FUNCTION_BLOCK FB_GroupElement_HMI EXTENDS FB_BaseGroupElement_HMI IMPLEMENTS ITF_GroupElement_HMI
VAR
	itfGroupElementConnector			: ITF_GroupElement_HMI_Connector;
	refstGroupElementData				: REFERENCE TO ST_GroupElement_HMI;
	
	itfControlElement1					: ITF_ControlElement_HMI;
	itfControlElement2					: ITF_ControlElement_HMI;
	itfComponent1						: ITF_Component_HMI;
	itfComponent2						: ITF_Component_HMI;
	
END_VAR

METHOD FB_init : BOOL
VAR_INPUT
	bInitRetains : BOOL; // if TRUE, the retain variables are initialized (warm start / cold start)
	bInCopyCode : BOOL;  // if TRUE, the instance afterwards gets moved into the copy code (online change)
	itfBaseLoggerConnector				: ITF_BaseLogger_HMI_Connector;	//bezpośredni łącznik do logera
	itfGroupElementConnector			: ITF_GroupElement_HMI_Init;
	itfControlElement1					: ITF_ControlElement_HMI;
	itfControlElement2					: ITF_ControlElement_HMI;
	itfComponent1						: ITF_Component_HMI;
	itfComponent2						: ITF_Component_HMI;
	
END_VAR
//Przypisanie do elementu który własnie stworzyliśmy
THIS^.itfGroupElementConnector			:= itfGroupElementConnector;
//Przypisanie do elementów z biblioteki
THIS^.itfBaseLoggerElementConnector		:= itfGroupElementConnector;
THIS^.itfBaseComponentConnector			:= itfGroupElementConnector;
THIS^.itfBaseControlElementConnector	:= itfGroupElementConnector;
THIS^.itfBaseGroupElementConnector		:= itfGroupElementConnector;
//
THIS^.itfBaseLoggerConnector			:= itfBaseLoggerConnector;
//
THIS^.itfControlElement1				:= itfControlElement1;
THIS^.itfControlElement2				:= itfControlElement2;
THIS^.itfComponent1						:= itfComponent1;
THIS^.itfComponent2						:= itfComponent2;

IF (THIS^.itfGroupElementConnector <> 0 AND
	THIS^.itfBaseLoggerElementConnector <> 0 AND
	THIS^.itfBaseComponentConnector	<> 0 AND
	THIS^.itfBaseControlElementConnector <> 0 AND
	THIS^.itfBaseGroupElementConnector <> 0 AND
	THIS^.itfBaseLoggerConnector <> 0) THEN
	THIS^.bIsInit						:= TRUE;
END_IF
END_METHOD

METHOD LinkGroupelementData : BOOL
VAR_INPUT
	stData					: REFERENCE TO ST_GroupElement_HMI_Link;
END_VAR
THIS^.refstGroupElementData	REF= stData.stGroupElement;

THIS^.refstBaseLoggerElementDataHMI	REF= stData.stBaseLoggerElement;
THIS^.refstBaseComponentDataHMI		REF= stData.stBaseComponent;
THIS^.refstBaseControlElementDataHMI	REF= stData.stBaseControlElement;
THIS^.refstBaseGroupElementDataHMI		REF= stData.stBaseGroupElement;

THIS^.itfControlElement1.LinkControlElementData (stData := stData.stControlElement1);
THIS^.itfControlElement2.LinkControlElementData (stData := stData.stControlElement2);
THIS^.itfComponent1.LinkComponentData (stData := stData.stComponent1);
THIS^.itfComponent2.LinkComponentData (stData := stData.stComponent2);

THIS^.CreateLinkToEventsMemory ();

IF (__ISVALIDREF (THIS^.refstGroupElementData) AND
	__ISVALIDREF (THIS^.refstBaseLoggerElementDataHMI) AND
	__ISVALIDREF (THIS^.refstBaseComponentDataHMI) AND
	__ISVALIDREF (THIS^.refstBaseControlElementDataHMI) AND
	__ISVALIDREF (THIS^.refstBaseGroupElementDataHMI)) THEN
	THIS^.bIsValidData		:= TRUE;
	LinkGroupelementData	:= TRUE;
END_IF
END_METHOD

END_FUNCTION_BLOCK

(* stored: Version 1.1.0.1, ProductVersion 3.1.4024.15
   POU FB_GroupElement_HMI: Id {19883d18-afce-4591-ab72-0deda3f3642e}, SpecialFunc None
   Folder ITF_GroupElement_HMI: Id {c7262793-080a-4a80-b8cd-5912156ea0a0}
   Method FB_init: Id {60cf9aa3-a3c1-477d-943b-0793fbe6bf08}
   Method LinkGroupelementData: Id {a9cd9d23-e72d-4255-8d5b-60aaf945db36} *)
